// TIA Portal V18 export
// export: Created 2026-03-12T16:04:35.3963979Z, ExportSetting WithDefaults, DisplayName Totally Integrated Automation Portal, DisplayVersion V18 Update 5, DisplayName TIA Portal Openness, DisplayVersion V18 Update 5, DisplayName TIA Portal Version Control Interface, DisplayVersion V18, DisplayName SINAMICS Startdrive Advanced, DisplayVersion V18, DisplayName SINAMICS Startdrive G130, G150, S120, S150, SINAMICS MV, S210, DisplayVersion V18, DisplayName SINAMICS Startdrive G110M, G120, G120C, G120D, G120P, G115D, DisplayVersion V18, DisplayName STEP 7 Professional, DisplayVersion V18 Update 5, DisplayName STEP 7 Safety, DisplayVersion V18, DisplayName WinCC Professional, DisplayVersion V18 Update 5
FUNCTION_BLOCK "FB VALVULA"   // FB17, LAD
{ S7_Optimized_Access := 'TRUE' }
VERSION : 0.1
// Network 1: Gerenciamento Status Válvula
// Network 2: Recebimento dos sinais de entrada (Sinais de campo e comandos)
// Network 3: MODO MANUAL: Conjunto de condições para ligar e desligar
// Network 4: MODO AUTOMÁTICO: Conjunto de condições para ligar e desligar
// Network 5: FALHA: Condicionamento de falha
// Network 6: LIGA BOMBA: Validando intertravamentos para ligar
// Network 7: ABRE VÁLVULA: Validando intertravamentos para abrir
// stored: AutoNumber true, IsIECCheckEnabled false, IsRetainMemResEnabled false, MemoryReserve 100, SetENOAutomatically false, UDAEnableTagReadback false
   VAR_INPUT
      INPUT_ABERTA : Bool;   // 1 = Sinal elétrico de campo indicando válvula aberta
      INPUT_FECHADA : Bool;   // 1 = Sinal elétrico de campo indicando válvula fechada
      INPUT_FALHA : Bool;   // 0 = Sinal elétrico de campo indicando válvula em falha
      INPUT_LOCAL : Bool;   // 1 = Sinal elétrico de campo indicando válvula em modo local
      INPUT_REMOTO : Bool;   // 1 = Sinal elétrico de campo indicando válvula em modo remoto
      INPUT_FALHA_PROFINET : Bool;   // 1 = Indica falta de comunicação PROFINET com o equipamento
      INPUT_LIGA_AUTO : Bool;   // 1= indica que o processo pode ser ligado remoto manual
      PARAMETRO_ABRE : Bool;   // Parâmetro utilizado para abrir a válvula em modo automático
      PARAMETRO_FECHA : Bool;   // Parâmetro utilizado para fechar a válvula em modo automático
      CMD_ABRE : Bool;   // Comando enviado da IHM/SCADA para abrir a válvula
      CMD_MANUTEN : Bool;   // Comando enviado da IHM/SCADA para colocar a válvula em Modo de Manutenção
      CMD_MODO : Bool;   // Comando enviado da IHM/SCADA para colocar a bomba em (0 = Modo Manual, 1 = Modo Automático)
   END_VAR
   VAR_OUTPUT
      STATUS_VALV : Byte;   // 0 = FECHADA; 1 = ABERTA; 2 = FALHA
      ABRE_VALVULA : Bool;   // Saída acionada para abrir a válvula remotamente
      FECHA_VALVULA : Bool;   // Saída acionada para fechar a válvula remotamente
      REMOTO_MAN : Bool;   // Modo de Operação Remoto Manual
      REMOTO_AUTO : Bool;   // Modo de Operação Remoto Automático
      LOCAL_MAN : Bool;   // Modo de Operação Local Manual
   END_VAR
   VAR
      MANUTEN : Bool;   // Variável local para Indicar bomba em Modo Manutenção
      REMOTO : Bool;   // Variável local para indicar Modo Remoto
      FALHA : Bool;   // Variável local para Válvula em Falha
      ABRE_REM_MAN : Bool;   // Variável local para Acionamento Remoto Manual
      ABRE_REM_AUTO : Bool;   // Variável local para Acionamento Remoto Automático
   END_VAR
   VAR_TEMP   // added for the SCL form of the ladder/FBD networks
      _w1 : Bool;
   END_VAR
BEGIN

REGION Network 1: Gerenciamento Status Válvula
   // INPUT_ABERTA = Entrada de sinal de Válvula Aberta
   // INPUT_FECHADA = Entrada de sinal de Válvula Fechada
   // INPUT_FALHA = Entrada de sinal de Válvula em Falha
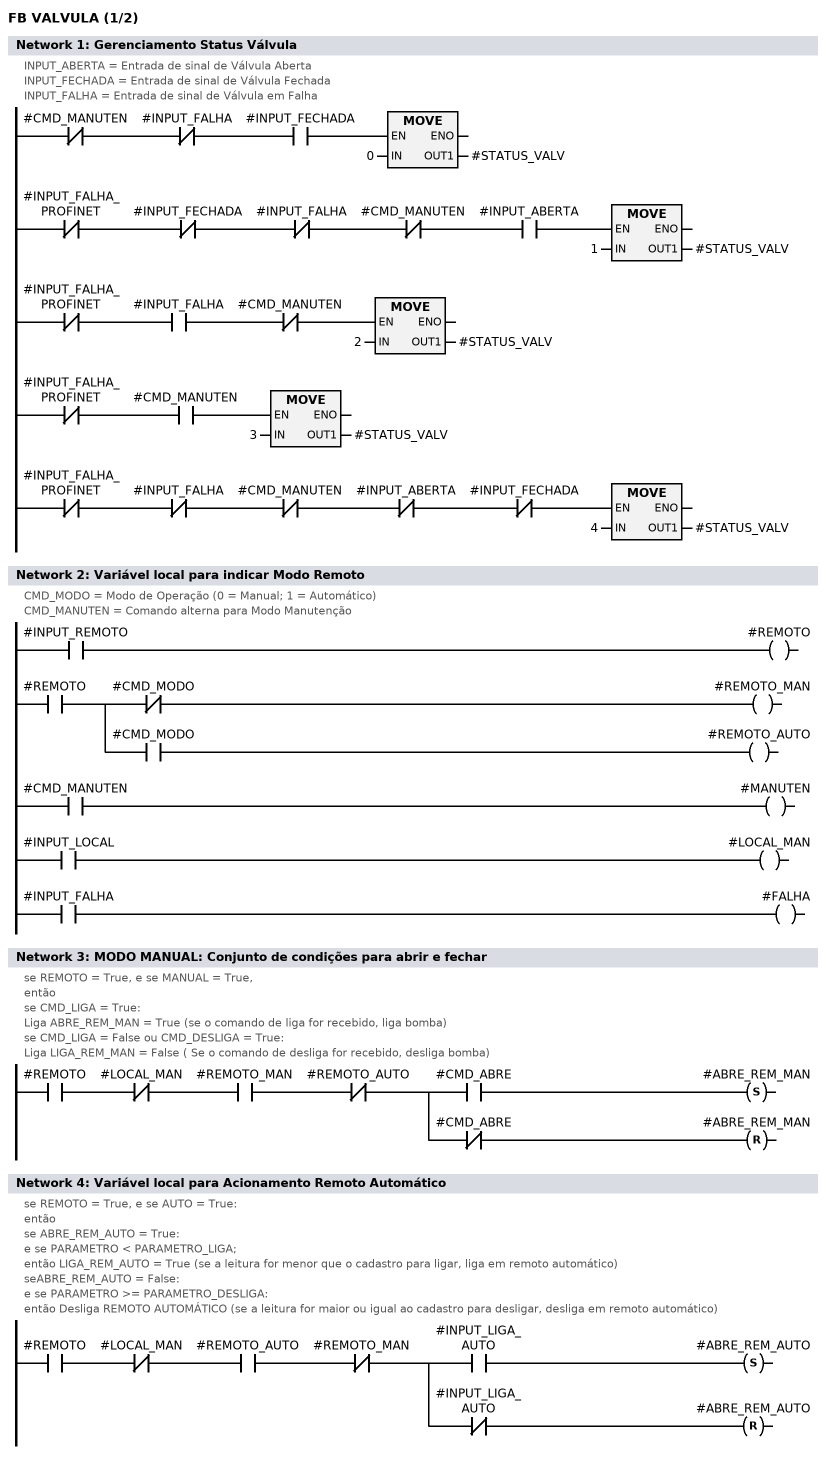
   RUNG wire#powerrail
      I_Contact( #CMD_MANUTEN )
      I_Contact( #INPUT_FALHA )
      Contact( #INPUT_FECHADA )
      Move(in := 0, out1 => #STATUS_VALV)
   END_RUNG
   RUNG wire#powerrail
      I_Contact( #INPUT_FALHA_PROFINET )
      I_Contact( #INPUT_FECHADA )
      I_Contact( #INPUT_FALHA )
      I_Contact( #CMD_MANUTEN )
      Contact( #INPUT_ABERTA )
      Move(in := 1, out1 => #STATUS_VALV)
   END_RUNG
   RUNG wire#powerrail
      I_Contact( #INPUT_FALHA_PROFINET )
      Contact( #INPUT_FALHA )
      I_Contact( #CMD_MANUTEN )
      Move(in := 2, out1 => #STATUS_VALV)
   END_RUNG
   RUNG wire#powerrail
      I_Contact( #INPUT_FALHA_PROFINET )
      Contact( #CMD_MANUTEN )
      Move(in := 3, out1 => #STATUS_VALV)
   END_RUNG
   RUNG wire#powerrail
      I_Contact( #INPUT_FALHA_PROFINET )
      I_Contact( #INPUT_FALHA )
      I_Contact( #CMD_MANUTEN )
      I_Contact( #INPUT_ABERTA )
      I_Contact( #INPUT_FECHADA )
      Move(in := 4, out1 => #STATUS_VALV)
   END_RUNG
   // the same network as SCL:
   IF NOT #CMD_MANUTEN AND NOT #INPUT_FALHA AND #INPUT_FECHADA THEN #STATUS_VALV := 0; END_IF;
   IF NOT #INPUT_FALHA_PROFINET AND NOT #INPUT_FECHADA AND NOT #INPUT_FALHA AND NOT #CMD_MANUTEN AND #INPUT_ABERTA THEN
       #STATUS_VALV := 1;
   END_IF;
   IF NOT #INPUT_FALHA_PROFINET AND #INPUT_FALHA AND NOT #CMD_MANUTEN THEN #STATUS_VALV := 2; END_IF;
   IF NOT #INPUT_FALHA_PROFINET AND #CMD_MANUTEN THEN #STATUS_VALV := 3; END_IF;
   IF NOT #INPUT_FALHA_PROFINET AND NOT #INPUT_FALHA AND NOT #CMD_MANUTEN AND NOT #INPUT_ABERTA AND NOT #INPUT_FECHADA THEN
       #STATUS_VALV := 4;
   END_IF;
END_REGION

REGION Network 2: Variável local para indicar Modo Remoto
   // CMD_MODO = Modo de Operação (0 = Manual; 1 = Automático)
   // CMD_MANUTEN = Comando alterna para Modo Manutenção
   RUNG wire#powerrail
      Contact( #INPUT_REMOTO )
      Coil( #REMOTO )
   END_RUNG
   RUNG wire#powerrail
      Contact( #REMOTO )
      wire#w1
      I_Contact( #CMD_MODO )
      Coil( #REMOTO_MAN )
   END_RUNG
   RUNG wire#w1
      Contact( #CMD_MODO )
      Coil( #REMOTO_AUTO )
   END_RUNG
   RUNG wire#powerrail
      Contact( #CMD_MANUTEN )
      Coil( #MANUTEN )
   END_RUNG
   RUNG wire#powerrail
      Contact( #INPUT_LOCAL )
      Coil( #LOCAL_MAN )
   END_RUNG
   RUNG wire#powerrail
      Contact( #INPUT_FALHA )
      Coil( #FALHA )
   END_RUNG
   // the same network as SCL:
   #REMOTO := #INPUT_REMOTO;
   #REMOTO_MAN := #REMOTO AND NOT #CMD_MODO;
   #REMOTO_AUTO := #REMOTO AND #CMD_MODO;
   #MANUTEN := #CMD_MANUTEN;
   #LOCAL_MAN := #INPUT_LOCAL;
   #FALHA := #INPUT_FALHA;
END_REGION

REGION Network 3: MODO MANUAL: Conjunto de condições para abrir e fechar
   // se REMOTO = True, e se MANUAL = True,
   // 
   // então
   // se CMD_LIGA = True: 
   // Liga ABRE_REM_MAN = True (se o comando de liga for recebido, liga bomba)
   // 
   // se CMD_LIGA = False ou CMD_DESLIGA = True:
   // Liga LIGA_REM_MAN = False ( Se o comando de desliga for recebido, desliga bomba)
   RUNG wire#powerrail
      Contact( #REMOTO )
      I_Contact( #LOCAL_MAN )
      Contact( #REMOTO_MAN )
      I_Contact( #REMOTO_AUTO )
      wire#w1
      Contact( #CMD_ABRE )
      S_Coil( #ABRE_REM_MAN )
   END_RUNG
   RUNG wire#w1
      I_Contact( #CMD_ABRE )
      R_Coil( #ABRE_REM_MAN )
   END_RUNG
   // the same network as SCL:
   #_w1 := #REMOTO AND NOT #LOCAL_MAN AND #REMOTO_MAN AND NOT #REMOTO_AUTO;
   IF #_w1 AND #CMD_ABRE THEN #ABRE_REM_MAN := TRUE; END_IF;
   IF #_w1 AND NOT #CMD_ABRE THEN #ABRE_REM_MAN := FALSE; END_IF;
END_REGION

REGION Network 4: Variável local para Acionamento Remoto Automático
   // se REMOTO = True, e se AUTO = True:
   // 
   // então
   // se ABRE_REM_AUTO = True:
   // e se PARAMETRO < PARAMETRO_LIGA;
   // então LIGA_REM_AUTO = True (se a leitura for menor que o cadastro para ligar, liga em remoto automático)
   // 
   // seABRE_REM_AUTO = False:
   // e se PARAMETRO >= PARAMETRO_DESLIGA:
   // então Desliga REMOTO AUTOMÁTICO (se a leitura for maior ou igual ao cadastro para desligar, desliga em remoto automático)
   RUNG wire#powerrail
      Contact( #REMOTO )
      I_Contact( #LOCAL_MAN )
      Contact( #REMOTO_AUTO )
      I_Contact( #REMOTO_MAN )
      wire#w1
      Contact( #INPUT_LIGA_AUTO )
      S_Coil( #ABRE_REM_AUTO )
   END_RUNG
   RUNG wire#w1
      I_Contact( #INPUT_LIGA_AUTO )
      R_Coil( #ABRE_REM_AUTO )
   END_RUNG
   // the same network as SCL:
   #_w1 := #REMOTO AND NOT #LOCAL_MAN AND #REMOTO_AUTO AND NOT #REMOTO_MAN;
   IF #_w1 AND #INPUT_LIGA_AUTO THEN #ABRE_REM_AUTO := TRUE; END_IF;
   IF #_w1 AND NOT #INPUT_LIGA_AUTO THEN #ABRE_REM_AUTO := FALSE; END_IF;
END_REGION

REGION Network 5: FALHA: Condicionamento de falha
   // se FALHA = False;
   // 
   // então
   // ABRE_REM_AUTO = False (Reseta Liga Remoto Automático)
   // ABRE_REM_MAN = False (Reseta Liga Remoto Manual)
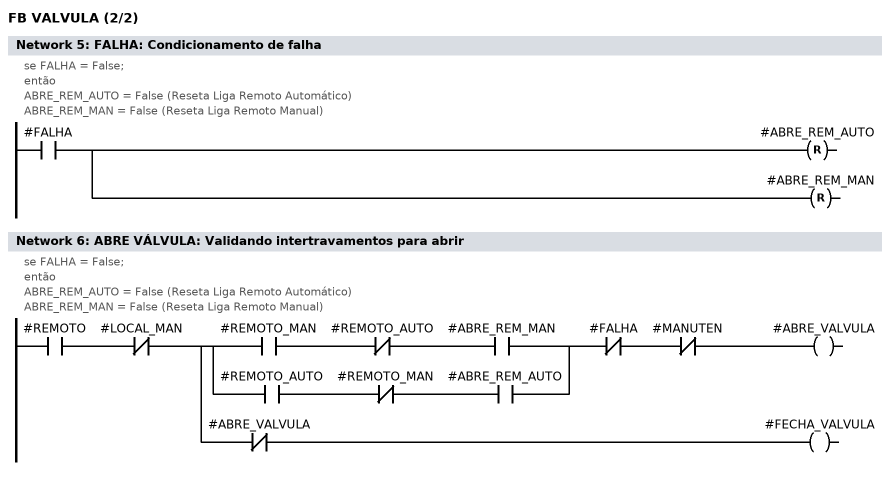
   RUNG wire#powerrail
      Contact( #FALHA )
      wire#w1
      R_Coil( #ABRE_REM_AUTO )
   END_RUNG
   RUNG wire#w1
      R_Coil( #ABRE_REM_MAN )
   END_RUNG
   // the same network as SCL:
   IF #FALHA THEN
       #ABRE_REM_AUTO := FALSE;
       #ABRE_REM_MAN := FALSE;
   END_IF;
END_REGION

REGION Network 6: ABRE VÁLVULA: Validando intertravamentos para abrir
   // se FALHA = False;
   // 
   // então
   // ABRE_REM_AUTO = False (Reseta Liga Remoto Automático)
   // ABRE_REM_MAN = False (Reseta Liga Remoto Manual)
   RUNG wire#powerrail
      Contact( #REMOTO )
      I_Contact( #LOCAL_MAN )
      wire#w1
      Contact( #REMOTO_MAN )
      I_Contact( #REMOTO_AUTO )
      Contact( #ABRE_REM_MAN )
      wire#w2
      I_Contact( #FALHA )
      I_Contact( #MANUTEN )
      Coil( #ABRE_VALVULA )
   END_RUNG
   RUNG wire#w1
      Contact( #REMOTO_AUTO )
      I_Contact( #REMOTO_MAN )
      Contact( #ABRE_REM_AUTO )
   END_RUNG wire#w2
   RUNG wire#w1
      I_Contact( #ABRE_VALVULA )
      Coil( #FECHA_VALVULA )
   END_RUNG
   // the same network as SCL:
   #_w1 := #REMOTO AND NOT #LOCAL_MAN;
   #ABRE_VALVULA := #_w1 AND ((#REMOTO_MAN AND NOT #REMOTO_AUTO AND #ABRE_REM_MAN) OR (#REMOTO_AUTO AND NOT #REMOTO_MAN AND #ABRE_REM_AUTO)) AND NOT #FALHA AND NOT #MANUTEN;
   #FECHA_VALVULA := #_w1 AND NOT #ABRE_VALVULA;
END_REGION
END_FUNCTION_BLOCK
